FUNCTION_BLOCK ActivateProcess EXTENDS BaseProcess
VAR_INPUT
END_VAR
VAR_OUTPUT
END_VAR
VAR_IN_OUT
END_VAR
VAR
	///At least 1 variable needed because subclass members of an empty class are not exposed by OPC UA (TwinCAT bug!)
	{attribute 'OPC.UA.DA' := '0'}
	testVar: BOOL;
END_VAR

IF do_request THEN
    do_request_result := request();
    do_request := FALSE;
END_IF;
SUPER^();

{attribute 'TcRpcEnable' := '1'}
METHOD request : RequestResults
VAR_INPUT
END_VAR
VAR_OUTPUT
END_VAR
VAR_IN_OUT
END_VAR
VAR
END_VAR
IF THIS^.statuses.enabledStatus.enabled THEN
    THIS^.start();
    request := RequestResults.ACCEPTED;
ELSE
    request := RequestResults.REJECTED;
END_IF;
END_METHOD

{attribute 'TcRpcEnable' := '1'}
METHOD start
VAR_INPUT
END_VAR
VAR_OUTPUT
END_VAR
VAR_IN_OUT
END_VAR
VAR
END_VAR
THIS^.statuses.busyStatus( isBusy := TRUE );
THIS^.statuses.healthStatus( isGood := TRUE );
END_METHOD

END_FUNCTION_BLOCK

(* stored: Version 1.1.0.1, ProductVersion 3.1.4019.2
   POU ActivateProcess: Id {c2710e1a-578e-4fa4-be7b-d854762efbc8}, SpecialFunc None
   Method request: Id {1847e746-663b-4193-ba96-cbb03741fdd9}
   Method start: Id {62a21086-4a5b-4868-9cd4-fb27abac38ee} *)
